(* IEC 61131-3 sources: repolevel_ST_code_completion/output/0121完整版本/repoeval_elevator/readful_result_no_provide, 5 files *)

(* ---- F_DetectCurrentFloor.st ---- *)
IF FloorSensor0 THEN
	F_DetectCurrentFloor := 0;
ELSIF FloorSensor1 THEN
	F_DetectCurrentFloor := 1;
ELSIF FloorSensor2 THEN
	F_DetectCurrentFloor := 2;
ELSIF FloorSensor3 THEN
	F_DetectCurrentFloor := 3;
ELSE
	F_DetectCurrentFloor := CurrentFloor;
END_IF;
RETURN;
END_FUNCTION

(* ---- F_RegisterCalls.st ---- *)
IF CallGround THEN
  TargetFloors[0] := TRUE; // Assign TRUE to the 0th index if CallGround is triggered
END_IF;

IF CallFloor1 THEN
  TargetFloors[1] := TRUE; // Assign TRUE to the 1st index if CallFloor1 is triggered
END_IF;

IF CallFloor2 THEN
  TargetFloors[2] := TRUE; // Assign TRUE to the 2nd index if CallFloor2 is triggered
END_IF;

IF CallFloor3 THEN
  TargetFloors[3] := TRUE; // Assign TRUE to the 3rd index if CallFloor3 is triggered
END_IF;

RETURN // Correctly terminate the FUNCTION without a trailing semicolon after RETURN
END_FUNCTION

(* ---- F_UpdateDoorAnimation.st ---- *)
VAR
	nNewAni			:	DINT;		// 新的动画值
END_VAR

nNewAni := nCurrentAni;

// 开门动画（增加动画值）
IF bOpenDoor AND nNewAni < nMaxAni AND bCallFloor THEN
	nNewAni := nNewAni + 1;
END_IF

// 关门动画（减少动画值）
IF bCloseDoor AND nNewAni > 0 THEN
	nNewAni := nNewAni - 1;
END_IF

F_UpdateDoorAnimation := nNewAni;
RETURN;
END_FUNCTION

(* ---- FB_ElevatorDoorController.st ---- *)
VAR
	fbDoorTimer			:	TON;		// 开门延时定时器
	fbCloseDoorTimer	:	TON;		// 关门延时定时器
	nState				:	INT;		// 状态机
END_VAR

CASE nState OF
	0: // 空闲状态
		bOpenDoor := FALSE;
		bCloseDoor := FALSE;
		bDoorReady := TRUE;

		IF bArrivedAtTarget THEN
			nState := 1; // 开始开门流程
		END_IF

	1: // 开门延时
		bCloseDoor := FALSE;
		bDoorReady := FALSE;
		fbDoorTimer(IN := TRUE, PT := T#2S);

		IF fbDoorTimer.Q THEN
			fbDoorTimer(IN := FALSE);
			nState := 2;
		END_IF

	2: // 开门
		bOpenDoor := TRUE;
		bDoorOpen := TRUE;
		bDoorReady := FALSE;

		IF NOT bArrivedAtTarget THEN
			nState := 3; // 开始关门流程
		END_IF

	3: // 关门延时
		bOpenDoor := FALSE;
		bDoorOpen := FALSE;
		bDoorReady := FALSE;
		fbCloseDoorTimer(IN := TRUE, PT := T#2S);

		IF fbCloseDoorTimer.Q THEN
			fbCloseDoorTimer(IN := FALSE);
			nState := 4;
		END_IF

	4: // 关门
		bCloseDoor := TRUE;
		bDoorReady := FALSE;

		IF bDoorClosed THEN
			bCloseDoor := FALSE;
			bDoorReady := TRUE;
			nState := 0; // 返回空闲状态
		END_IF

ELSE
	nState := 0; // 默认返回空闲状态
END_CASE
END_FUNCTION_BLOCK

(* ---- FB_ElevatorMovement.st ---- *)
VAR
	fbMoveDelayTimer	:	TON;				// 移动延时定时器
	i					:	INT;				// 循环变量
	bHasUpperRequest	:	BOOL;				// 有更高楼层请求
	bHasLowerRequest	:	BOOL;				// 有更低楼层请求
END_VAR

// 检查是否到达目标楼层
IF TargetFloors[CurrentFloor] THEN
	bArrivedAtTarget := TRUE;
	TargetFloors[CurrentFloor] := FALSE; // 清除请求
	bMovingUp := FALSE;
	bMovingDown := FALSE;
	RETURN;
ELSE
	bArrivedAtTarget := FALSE;
END_IF

// 检查是否有更高楼层请求
bHasUpperRequest := FALSE;
FOR i := CurrentFloor + 1 TO 3 DO
	IF TargetFloors[i] THEN
		bHasUpperRequest := TRUE;
		EXIT;
	END_IF
END_FOR

// 检查是否有更低楼层请求
bHasLowerRequest := FALSE;
FOR i := CurrentFloor - 1 TO 0 BY -1 DO
	IF TargetFloors[i] THEN
		bHasLowerRequest := TRUE;
		EXIT;
	END_IF
END_FOR

// 控制电梯移动方向
IF bDoorReady THEN
	IF bHasUpperRequest THEN
		bMovingUp := TRUE;
		bMovingDown := FALSE;
	ELSIF bHasLowerRequest THEN
		bMovingUp := FALSE;
		bMovingDown := TRUE;
	ELSE
		bMovingUp := FALSE;
		bMovingDown := FALSE;
	END_IF
END_IF
END_FUNCTION_BLOCK
